(* PLC project SafeLOGIC-1, BrAutomation SafeDESIGNER  4.4.0.0 *)
(* stored: companyURL http://www.br-automation.com, creationDateTime Thu Aug 19 09:55:15 2021 *)

PROGRAM Main

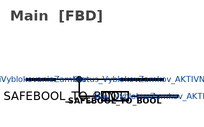
(* FBD diagram, written out as Structured Text *)
Status_VyblokovZamkov_AKTIVNE := siVyblokovanieZamkov;
Stav_VyblokovZamkov_AKTIVNE := SAFEBOOL_TO_BOOL(siVyblokovanieZamkov);
END_PROGRAM
